// TIA Portal V19 program export: 1 tag tables, 1 data types, 1 data blocks, 6 code blocks (in call order from the OBs), 0 instance data blocks

VAR_GLOBAL   // PLC tag table "Test"
   bReset AT %I0.0 : Bool;
   bTestFirstScan AT %I0.1 : Bool;
   bTestMonthShift AT %I0.2 : Bool;
   bTEstREset AT %I0.3 : Bool;
END_VAR
VAR_GLOBAL CONSTANT   // user constants
   MAX_DAYS_IN_MONTH : Int := 31;
END_VAR

TYPE "array2Months"
   STRUCT
      Current : Array[1.."MAX_DAYS_IN_MONTH"] of Real;
      Last : Array[1.."MAX_DAYS_IN_MONTH"] of Real;
   END_STRUCT;
END_TYPE

DATA_BLOCK "Data"   // DB5
{ S7_Optimized_Access := 'TRUE' }
// stored: MemoryReserve 100
   VAR
      Second : Int;
      Day : Int;
      Mothercores { S7_SetPoint := 'True'} : "array2Months";
      setsProduced { S7_SetPoint := 'True'} : "array2Months";
   END_VAR
BEGIN
END_DATA_BLOCK

ORGANIZATION_BLOCK "Main"   // OB1, FBD, ProgramCycle
TITLE = "Main Program Sweep (Cycle)"
{ S7_Optimized_Access := 'TRUE' }
// stored: SetENOAutomatically false
   VAR_INPUT
      Initial_Call : Bool;   // Initial call of this OB
      Remanence : Bool;   // =True, if remanent data are available
   END_VAR
   VAR_TEMP   // added for the SCL form of the ladder/FBD networks
      _w1 : Bool;
   END_VAR
BEGIN

REGION Network 1
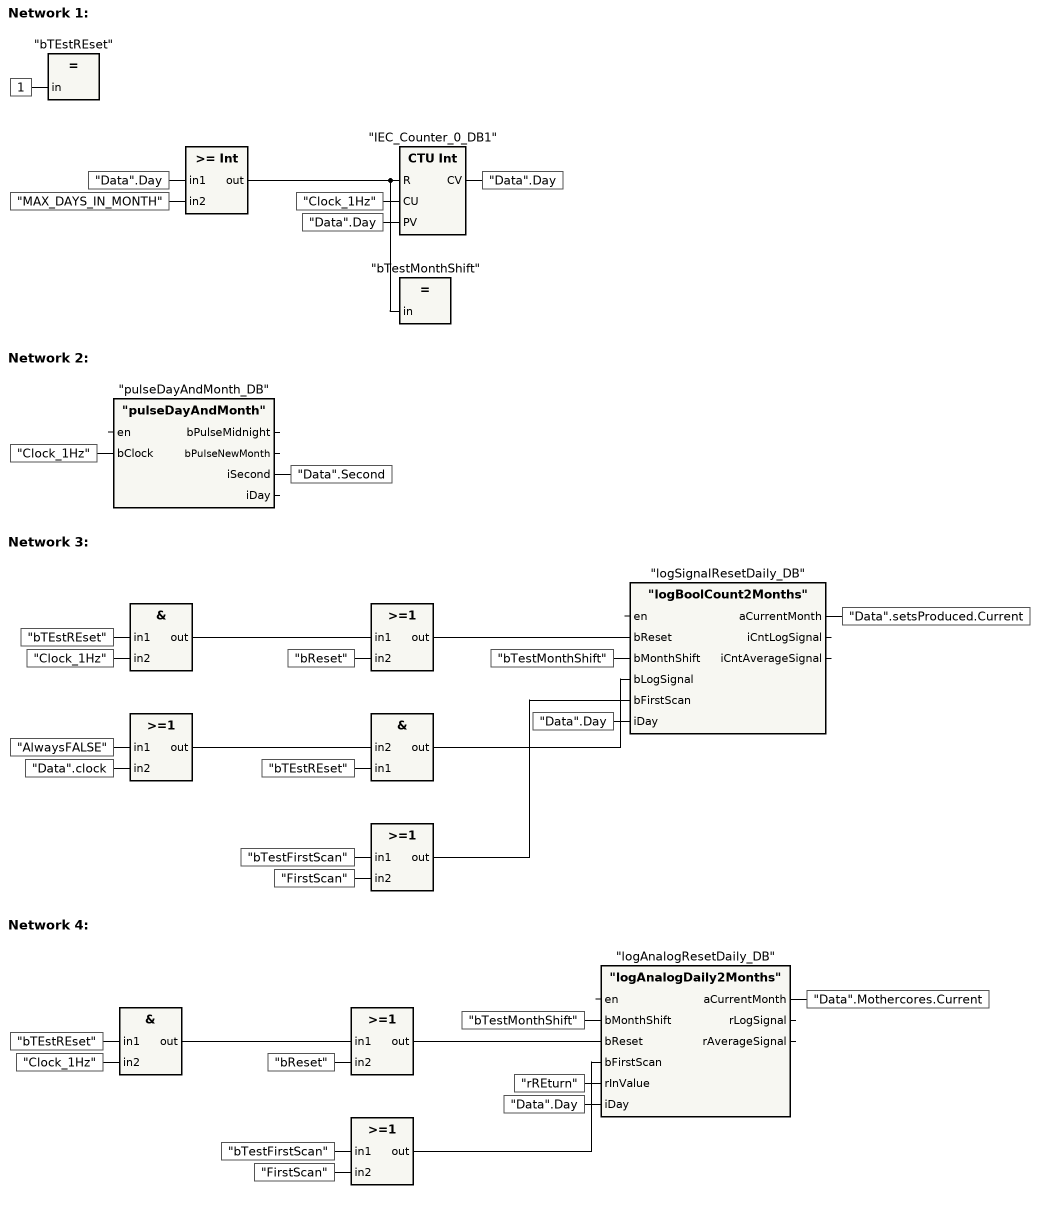
   "bTEstREset" := 1;
   #_w1 := "Data".Day >= "MAX_DAYS_IN_MONTH";
   "IEC_Counter_0_DB1".CTU(R := #_w1, CU := "Clock_1Hz", PV := "Data".Day, CV => "Data".Day);
   "bTestMonthShift" := #_w1;
END_REGION

REGION Network 2
   "pulseDayAndMonth_DB"(bClock := "Clock_1Hz", iSecond => "Data".Second);   // "pulseDayAndMonth"
END_REGION

REGION Network 3
   "logSignalResetDaily_DB"(bReset := ("bTEstREset" AND "Clock_1Hz") OR "bReset",   // "logBoolCount2Months"
                           bMonthShift := "bTestMonthShift",
                           bLogSignal := ("AlwaysFALSE" OR "Data".clock) AND "bTEstREset",
                           bFirstScan := "bTestFirstScan" OR "FirstScan",
                           iDay := "Data".Day,
                           aCurrentMonth => "Data".setsProduced.Current);
END_REGION

REGION Network 4
   "logAnalogResetDaily_DB"(bMonthShift := "bTestMonthShift",   // "logAnalogDaily2Months"
                           bReset := ("bTEstREset" AND "Clock_1Hz") OR "bReset",
                           bFirstScan := "bTestFirstScan" OR "FirstScan",
                           rInValue := "rREturn",
                           iDay := "Data".Day,
                           aCurrentMonth => "Data".Mothercores.Current);
END_REGION

REGION Network 5
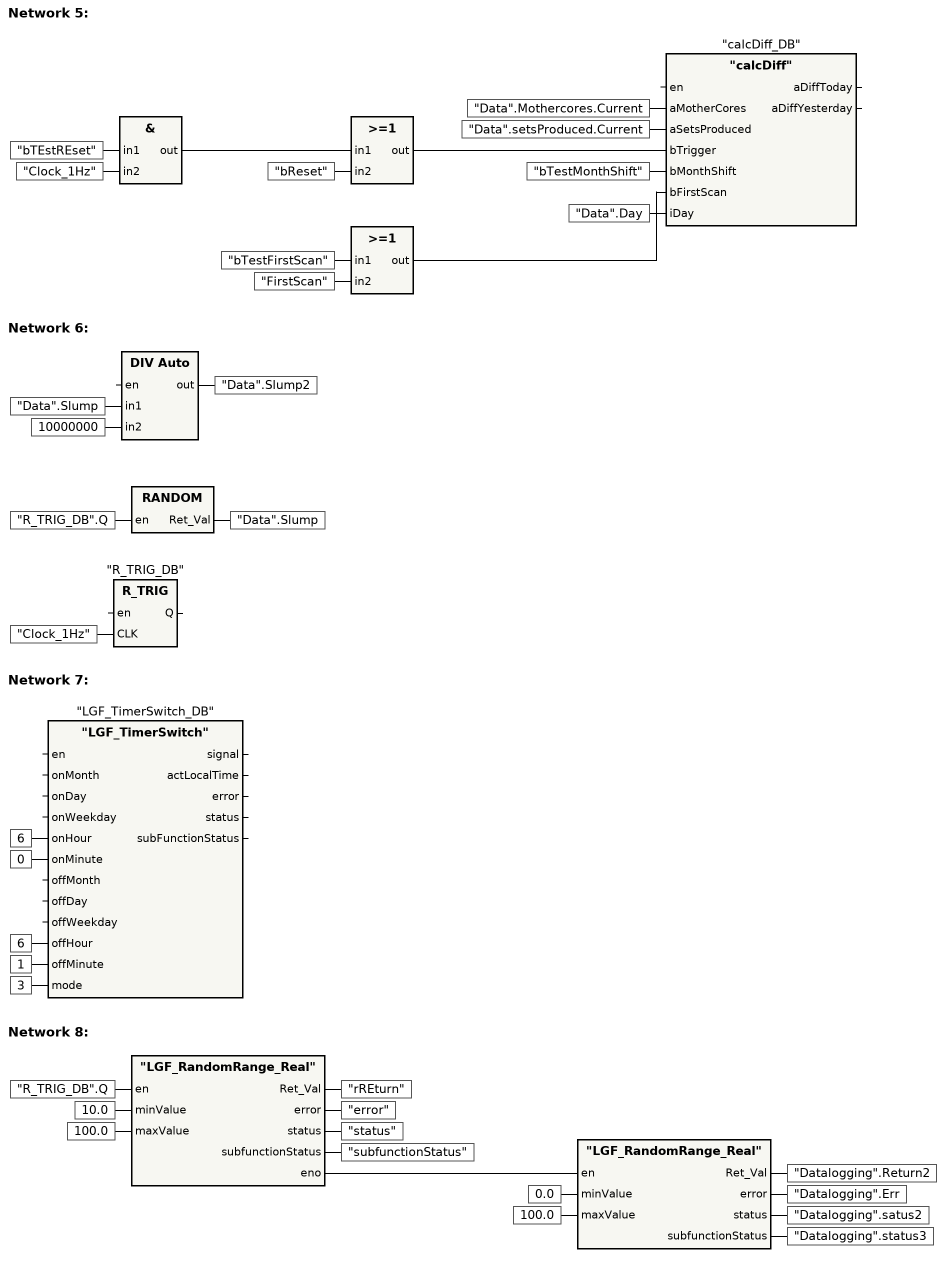
   "calcDiff_DB"(aMotherCores := "Data".Mothercores.Current,   // "calcDiff"
                 aSetsProduced := "Data".setsProduced.Current,
                 bTrigger := ("bTEstREset" AND "Clock_1Hz") OR "bReset",
                 bMonthShift := "bTestMonthShift",
                 bFirstScan := "bTestFirstScan" OR "FirstScan",
                 iDay := "Data".Day);
END_REGION

REGION Network 6
   "Data".Slump2 := "Data".Slump / 10000000;
   IF "R_TRIG_DB".Q THEN "Data".Slump := Random(); END_IF;
   "R_TRIG_DB"(CLK := "Clock_1Hz");   // R_TRIG
END_REGION

REGION Network 7
   "LGF_TimerSwitch_DB"(onHour := 6, onMinute := 0, offHour := 6, offMinute := 1, mode := 3);   // "LGF_TimerSwitch"
END_REGION

REGION Network 8
   "rREturn" := "LGF_RandomRange_Real"(EN := "R_TRIG_DB".Q,
                           minValue := 10.0,
                           maxValue := 100.0,
                           error => "error",
                           status => "status",
                           subfunctionStatus => "subfunctionStatus",
                           ENO => #_w1);
   IF #_w1 THEN
       "Datalogging".Return2 := "LGF_RandomRange_Real"(minValue := 0.0,
                               maxValue := 100.0,
                               error => "Datalogging".Err,
                               status => "Datalogging".satus2,
                               subfunctionStatus => "Datalogging".status3);
   END_IF;
END_REGION

REGION Network 9
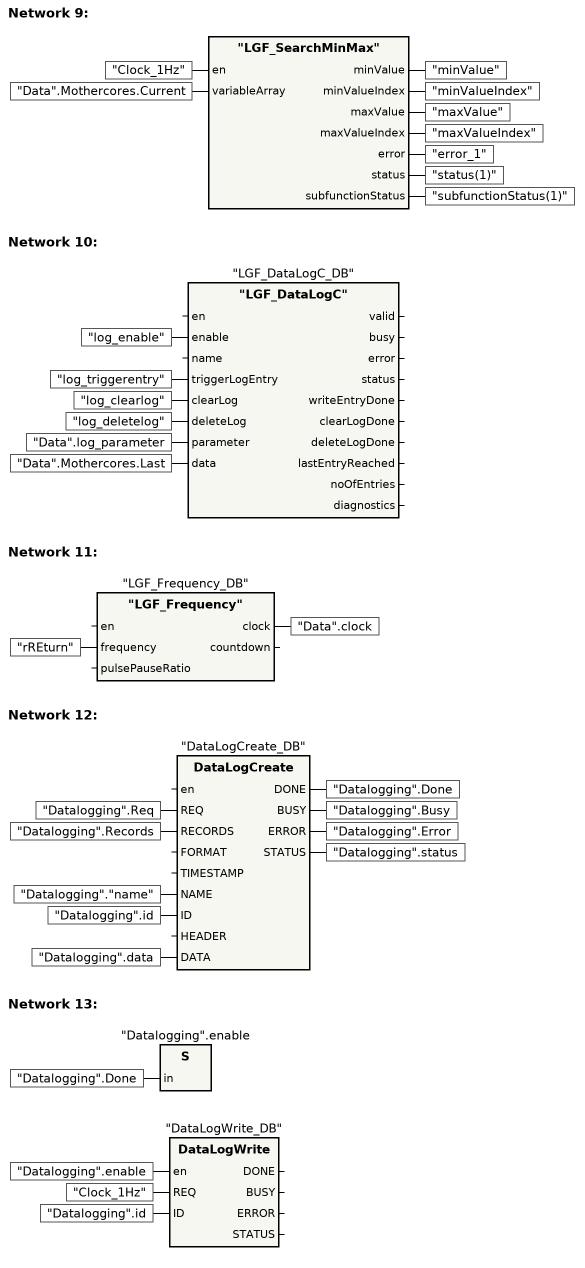
   IF "Clock_1Hz" THEN
       "LGF_SearchMinMax"(variableArray := "Data".Mothercores.Current,
                          minValue => "minValue",
                          minValueIndex => "minValueIndex",
                          maxValue => "maxValue",
                          maxValueIndex => "maxValueIndex",
                          error => "error_1",
                          status => "status(1)",
                          subfunctionStatus => "subfunctionStatus(1)");
   END_IF;
END_REGION

REGION Network 10
   "LGF_DataLogC_DB"(enable := "log_enable",   // "LGF_DataLogC"
                     triggerLogEntry := "log_triggerentry",
                     clearLog := "log_clearlog",
                     deleteLog := "log_deletelog",
                     parameter := "Data".log_parameter,
                     data := "Data".Mothercores.Last);
END_REGION

REGION Network 11
   "LGF_Frequency_DB"(frequency := "rREturn", clock => "Data".clock);   // "LGF_Frequency"
END_REGION

REGION Network 12
   "DataLogCreate_DB"(REQ := "Datalogging".Req,   // DataLogCreate
                      RECORDS := "Datalogging".Records,
                      "NAME" := "Datalogging"."name",
                      ID := "Datalogging".id,
                      DATA := "Datalogging".data,
                      DONE => "Datalogging".Done,
                      BUSY => "Datalogging".Busy,
                      ERROR => "Datalogging".Error,
                      STATUS => "Datalogging".status);
END_REGION

REGION Network 13
   IF "Datalogging".Done THEN "Datalogging".enable := TRUE; END_IF;
   IF "Datalogging".enable THEN
       "DataLogWrite_DB"(REQ := "Clock_1Hz", ID := "Datalogging".id);   // DataLogWrite
   END_IF;
END_REGION

REGION Network 14
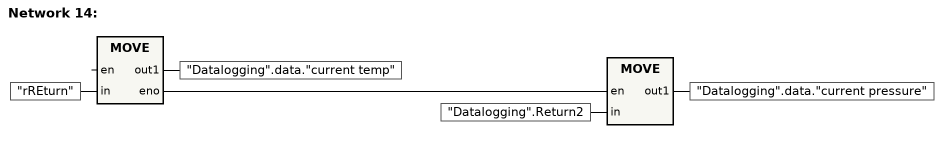
   "Datalogging".data."current temp" := "rREturn";
   "Datalogging".data."current pressure" := "Datalogging".Return2;
END_REGION
END_ORGANIZATION_BLOCK

FUNCTION_BLOCK "pulseDayAndMonth"
{ S7_Optimized_Access := 'TRUE' }
VERSION : 0.1
   VAR_INPUT 
      bClock : Bool;
   END_VAR

   VAR_OUTPUT 
      bPulseMidnight : Bool;
      bPulseNewMonth : Bool;
      iSecond : Int;
      iDay : Int;
   END_VAR

   VAR 
      R_TRIG_Midnight {InstructionName := 'R_TRIG'; LibVersion := '1.0'} : R_TRIG;
      R_TRIG_Month {InstructionName := 'R_TRIG'; LibVersion := '1.0'} : R_TRIG;
      R_TRIG_Second {InstructionName := 'R_TRIG'; LibVersion := '1.0'} : R_TRIG;
      NowTime {InstructionName := 'DTL'; LibVersion := '1.0'; S7_SetPoint := 'True'} : DTL;
      bClockPulse : Bool;
      iMonth : Int;
      iMonthMemory : Int;
      iHour : Int;
      iMinute : Int;
      bMidnight : Bool;
      bNewMonth : Bool;
      iTrigSecond { ExternalAccessible := 'False'; ExternalVisible := 'False'; ExternalWritable := 'False'} : Int := 1;
   END_VAR

   VAR_TEMP 
      iReturn : Int;
   END_VAR

   VAR CONSTANT 
      iTrigHour : Int := 6;
      iTrigMinute : Int := 0;
   END_VAR


BEGIN
	#R_TRIG_Second(CLK := #bClock,
	               Q => #bClockPulse);
	
	IF #bClockPulse THEN
	    #iReturn := RD_LOC_T(#NowTime);
	    #iMonth := #NowTime.MONTH;
	    #iDay := #NowTime.DAY;
	    #iHour := #NowTime.HOUR;
	    #iMinute := #NowTime.MINUTE;
	    #iSecond := #NowTime.SECOND;
	    
	    #bNewMonth := (#iMonth <> #iMonthMemory);
	    #iMonthMemory := #iMonth;
	    
	    #bMidnight := (#iHour = #iTrigHour AND #iMinute = #iTrigMinute AND #iSecond <= #iTrigSecond);
	END_IF;
	
	#R_TRIG_Midnight(CLK := #bMidnight,
	                 Q => #bPulseMidnight);
	#R_TRIG_Month(CLK := #bNewMonth,
	              Q => #bPulseNewMonth);
	
	
END_FUNCTION_BLOCK

FUNCTION_BLOCK "logBoolCount2Months"
{ S7_Optimized_Access := 'TRUE' }
VERSION : 0.1
   VAR_INPUT 
      bReset : Bool;
      bMonthShift : Bool;
      bLogSignal : Bool;
      bFirstScan : Bool;
      iDay : Int;
   END_VAR

   VAR_OUTPUT 
      aCurrentMonth : Array[1..#maxDays] of Real;
      iCntLogSignal : Real := 0.0;
      iCntAverageSignal : Real := 0.0;
   END_VAR

   VAR 
      R_TRIG_Signal {InstructionName := 'R_TRIG'; LibVersion := '1.0'} : R_TRIG;
   END_VAR
   VAR RETAIN
      IEC_Counter_Signal {InstructionName := 'CTU_INT'; LibVersion := '1.0'; ExternalAccessible := 'False'; ExternalVisible := 'False'; ExternalWritable := 'False'; S7_SetPoint := 'False'} : CTU_INT;
   END_VAR
   VAR 
      R_TRIG_Reset {InstructionName := 'R_TRIG'; LibVersion := '1.0'} : R_TRIG;
      aLastMonth : Array[1..#maxDays] of Real;
      i1 : Int;
      i2 : Int;
      i3 : Int;
      i4 : Int;
      R_TRIG_Month {InstructionName := 'R_TRIG'; LibVersion := '1.0'} : R_TRIG;
   END_VAR

   VAR CONSTANT 
      maxDays : Int := 31;
      maxCount : Int := 3000;
   END_VAR


BEGIN
	REGION Initialize
	    IF #bFirstScan THEN
	        #iCntLogSignal := 0.0;
	        #iCntAverageSignal := 0.0;
	        FOR #i4 := 1 TO #maxDays DO
	            #aCurrentMonth[#i4] := 0.0;
	            #aLastMonth[#i4] := 0.0;
	        END_FOR;
	    END_IF;
	END_REGION ;
	
	#R_TRIG_Reset(CLK := #bReset);
	#R_TRIG_Month(CLK := #bMonthShift);
	
	IF #R_TRIG_Reset.Q AND #iDay > 0 AND #iDay <= #maxDays THEN
	    
	    #aCurrentMonth[#iDay] := #iCntLogSignal;
	    #iCntAverageSignal := 0.0;
	    
	    FOR #i2 := 1 TO #maxDays BY 1 DO
	        #iCntAverageSignal := #iCntAverageSignal + #aCurrentMonth[#i2];
	    END_FOR;
	    #iCntAverageSignal := #iCntAverageSignal / (#maxDays);
	END_IF;
	
	REGION New month
	    IF #R_TRIG_Month.Q THEN
	        #aLastMonth := #aCurrentMonth;
	        FOR #i3 := 1 TO #maxDays BY 1 DO
	            #aCurrentMonth[#i3] := 0.0;
	        END_FOR;
	    END_IF;
	END_REGION
	
	#R_TRIG_Signal(CLK := #bLogSignal);
	
	#IEC_Counter_Signal(CU := #R_TRIG_Signal.Q,
	                    R := #R_TRIG_Reset.Q,
	                    PV := #maxCount,
	                    CV => #iCntLogSignal);
	
END_FUNCTION_BLOCK

FUNCTION_BLOCK "logAnalogDaily2Months"
{ S7_Optimized_Access := 'TRUE' }
VERSION : 0.1
   VAR_INPUT 
      bMonthShift : Bool;
      bReset : Bool;
      bFirstScan : Bool;
      rInValue : Real;
      iDay : Int;
   END_VAR

   VAR_OUTPUT RETAIN
      aCurrentMonth : Array[1..#maxDays] of Real;
   END_VAR
   VAR_OUTPUT 
      rLogSignal : Real;
      rAverageSignal : Real;
   END_VAR

   VAR 
      R_TRIG_Reset {InstructionName := 'R_TRIG'; LibVersion := '1.0'} : R_TRIG;
      R_TRIG_Month {InstructionName := 'R_TRIG'; LibVersion := '1.0'} : R_TRIG;
   END_VAR
   VAR RETAIN
      aLastMonth : Array[1..#maxDays] of Real;
   END_VAR
   VAR 
      i2 : Int;
      i3 : Int;
      i1 : Int;
   END_VAR

   VAR CONSTANT 
      maxDays : Int := 31;
   END_VAR


BEGIN
	//Sparar värdet av rLogSignal i aCurrentMonth under position för dagens datum, vid månadsskifte flyttas innehållet till aLastMonth och aCurrentMonth nollställs
	
	REGION Initialize
	    IF #bFirstScan THEN
	        #rLogSignal := 0.0;
	        #rAverageSignal := 0.0;
	        FOR #i1 := 1 TO #maxDays DO
	            #aCurrentMonth[#i1] := 0.0;
	            #aLastMonth[#i1] := 0.0;
	        END_FOR;
	    END_IF;
	END_REGION ;
	
	// Catch rising edges and create pulse
	#R_TRIG_Reset(CLK := #bReset);
	#R_TRIG_Month(CLK := #bMonthShift);
	
	
	REGION Store values in array at trigger
	    IF #R_TRIG_Reset.Q AND #iDay > 0 AND #iDay <= #maxDays THEN
	        #aCurrentMonth[#iDay] := #rInValue;
	        #rAverageSignal := 0.0;
	        
	        FOR #i2 := 1 TO #maxDays BY 1 DO //Calculate average signal
	            
	            #rAverageSignal := #rAverageSignal + #aCurrentMonth[#i2];
	            IF #aCurrentMonth[#i2] = 0 THEN
	                #rAverageSignal := #rAverageSignal / #i2;
	                EXIT;
	            END_IF;
	        END_FOR;
	        
	    END_IF;
	END_REGION 
	
	REGION New month
	    IF #R_TRIG_Month.Q THEN
	        #aLastMonth := #aCurrentMonth;
	        FOR #i3 := 1 TO #maxDays BY 1 DO
	            #aCurrentMonth[#i3] := 0.0;
	        END_FOR;
	    END_IF;
	END_REGION
	
	#rLogSignal := #rInValue;
	
END_FUNCTION_BLOCK

FUNCTION_BLOCK "calcDiff"
{ S7_Optimized_Access := 'TRUE' }
VERSION : 0.1
   VAR_INPUT 
      aMotherCores : Array[1..#daysLogged] of Real;
      aSetsProduced : Array[1..#daysLogged] of Real;
      bTrigger : Bool;
      bMonthShift : Bool;
      bFirstScan : Bool;
      iDay : Int;
   END_VAR

   VAR_OUTPUT 
      aDiffToday : Real;
      aDiffYesterday : Real;
   END_VAR

   VAR 
      aDifferenceCurrentLast : Array[1..#daysLogged] of Real;
      aDifferenceCurrent : Array[1..#daysLogged] of Real;
      R_TRIG_Reset {InstructionName := 'R_TRIG'; LibVersion := '1.0'} : R_TRIG;
      R_TRIG_Month {InstructionName := 'R_TRIG'; LibVersion := '1.0'} : R_TRIG;
      i3 : Int;
      i4 : Int;
   END_VAR

   VAR_TEMP 
      itempStorage : Real;
   END_VAR

   VAR CONSTANT 
      daysLogged : Int := 31;
   END_VAR


BEGIN
	REGION Initialize
	    IF #bFirstScan THEN
	        FOR #i4 := 1 TO #daysLogged DO
	            #aDifferenceCurrent[#i4] := 0.0;
	            #aDifferenceCurrentLast[#i4] := 0.0;
	        END_FOR;
	    END_IF;
	END_REGION ;
	
	#R_TRIG_Reset(CLK := #bTrigger);
	#R_TRIG_Month(CLK := #bMonthShift);
	
	REGION Loop log values
	    IF #R_TRIG_Reset.Q AND #iDay > 0 AND #iDay <= #daysLogged THEN
	        IF #aSetsProduced[#iDay] <> 0 AND #aMotherCores[#iDay] <> 0 THEN
	            //#aDifferenceCurrent[#iDay] := #aSetsProduced[#iDay] / #aMotherCores[#iDay];
	            #itempStorage := (ROUND(IN := 100 * (#aSetsProduced[#iDay] / #aMotherCores[#iDay])));
	            #aDifferenceCurrent[#iDay] := #itempStorage / 100;
	            //#aDifferenceCurrent[#iDay] := ROUND(IN := 100 * (#aSetsProduced[#iDay] / #aMotherCores[#iDay]))/100;
	        END_IF;
	    END_IF;
	END_REGION
	
	REGION New month
	    IF #R_TRIG_Month.Q THEN
	        #aDifferenceCurrentLast := #aDifferenceCurrent;
	        FOR #i3 := 1 TO #daysLogged BY 1 DO
	            #aDifferenceCurrent[#i3] := 0.0;
	        END_FOR;
	    END_IF;
	END_REGION
	
	IF #iDay <> 0 AND #iDay <= 31 THEN
	    #aDiffToday := #aDifferenceCurrent[#iDay];
	    
	    IF #iDay > 1 THEN
	        #aDiffYesterday := #aDifferenceCurrent[#iDay - 1];
	    ELSIF #iDay = 1 THEN
	        #aDiffYesterday := #aDifferenceCurrent[#iDay + 30];
	    END_IF;
	END_IF;
	
END_FUNCTION_BLOCK

FUNCTION_BLOCK "logAnalogDaily12Months"
{ S7_Optimized_Access := 'TRUE' }
VERSION : 0.1
   VAR_INPUT 
      bMonthShift : Bool;
      bReset : Bool;
      bFirstScan : Bool;
      rInValue : Real;
      iDay : Int;
   END_VAR

   VAR_OUTPUT RETAIN
      aCurrentMonth : Array[1..#maxDays] of Real;
   END_VAR
   VAR_OUTPUT 
      rLogSignal : Real;
      rAverageSignal : Real;
   END_VAR

   VAR 
      R_TRIG_Reset {InstructionName := 'R_TRIG'; LibVersion := '1.0'} : R_TRIG;
      R_TRIG_Month {InstructionName := 'R_TRIG'; LibVersion := '1.0'} : R_TRIG;
   END_VAR
   VAR RETAIN
      aLastMonth : Array[1..#maxDays] of Real;
   END_VAR
   VAR 
      i2 : Int;
      i3 : Int;
      i1 : Int;
   END_VAR

   VAR CONSTANT 
      maxDays : Int := 31;
   END_VAR


BEGIN
	//Sparar värdet av rLogSignal i aCurrentMonth under position för dagens datum, vid månadsskifte flyttas innehållet till aLastMonth och aCurrentMonth nollställs
	
	REGION Initialize
	    IF #bFirstScan THEN
	        #rLogSignal := 0.0;
	        #rAverageSignal := 0.0;
	        FOR #i1 := 1 TO #maxDays DO
	            #aCurrentMonth[#i1] := 0.0;
	            #aLastMonth[#i1] := 0.0;
	        END_FOR;
	    END_IF;
	END_REGION ;
	
	// Catch rising edges and create pulse
	#R_TRIG_Reset(CLK := #bReset);
	#R_TRIG_Month(CLK := #bMonthShift);
	
	
	REGION Store values in array at trigger
	    IF #R_TRIG_Reset.Q AND #iDay > 0 AND #iDay <= #maxDays THEN
	        #aCurrentMonth[#iDay] := #rInValue;
	        #rAverageSignal := 0.0;
	        
	        FOR #i2 := 1 TO #maxDays BY 1 DO //Calculate average signal
	            
	            #rAverageSignal := #rAverageSignal + #aCurrentMonth[#i2];
	            IF #aCurrentMonth[#i2] = 0 THEN
	                #rAverageSignal := #rAverageSignal / #i2;
	                EXIT;
	            END_IF;
	        END_FOR;
	        
	    END_IF;
	END_REGION 
	
	REGION New month
	    IF #R_TRIG_Month.Q THEN
	        #aLastMonth := #aCurrentMonth;
	        FOR #i3 := 1 TO #maxDays BY 1 DO
	            #aCurrentMonth[#i3] := 0.0;
	        END_FOR;
	    END_IF;
	END_REGION
	
	#rLogSignal := #rInValue;
	
END_FUNCTION_BLOCK
